Fanuc TP program (LS listing): mv_place.ls

/PROG MV_PLACE
/ATTR
DEFAULT_GROUP	= 1,*,*,*,*;
/MN
 : UFRAME_NUM=2 ;
 : UTOOL_NUM=2 ;
 : J PR[21:PLACE] 500% CNT100 Tool_Offset,PR[22:PLACE_APTO] ;
 : L PR[21:PLACE] 250mm/sec CNT0 ;
/POS
/END
